DATA_BLOCK "ST10_Flow5_FRobot_1_iDB"
{ S7_Optimized_Access := 'TRUE' }
VERSION : 0.1
NON_RETAIN
"ST10_Flow5_FRobot_1"

BEGIN

END_DATA_BLOCK

